// TIA Portal V17 export
// export: Created 2025-03-05T08:01:21.5015692Z, ExportSetting WithDefaults, DisplayName Totally Integrated Automation Portal, DisplayVersion V17 Update 8, DisplayName TIA Portal Openness, DisplayVersion V17 Update 8, DisplayName TIA Portal Version Control Interface, DisplayVersion V17, DisplayName SINAMICS Startdrive Advanced, DisplayVersion V17 SP2, DisplayName SINAMICS Startdrive G110M, G120, G120C, G120D, G120P, G115D, DisplayVersion V17 SP2, DisplayName SINAMICS Startdrive G130, G150, S120, S150, SINAMICS MV, S210, DisplayVersion V17 SP2, DisplayName STEP 7 Professional, DisplayVersion V17 Update 8, DisplayName SINUMERIK ONE STEP 7 Toolbox, DisplayVersion V17 Update 12, DisplayName SINUMERIK 840D sl STEP 7 Toolbox, DisplayVersion V17 Update 12, DisplayName STEP 7 Safety, DisplayVersion V17 Update 6, DisplayName WinCC Advanced, DisplayVersion V17 Update 8
FUNCTION "FC20202_LASER_TRUMPF_ACTIVE" : Void   // FC20202, LAD
TITLE = FC20202 LASER TRUMPF ACTIVE
{ S7_Optimized_Access := 'TRUE' }
VERSION : 0.1
// stored: AutoNumber false, IsIECCheckEnabled false, SetENOAutomatically false, UDAEnableTagReadback false
BEGIN

REGION Network 1: LASER UNIT 1 ACTIVE
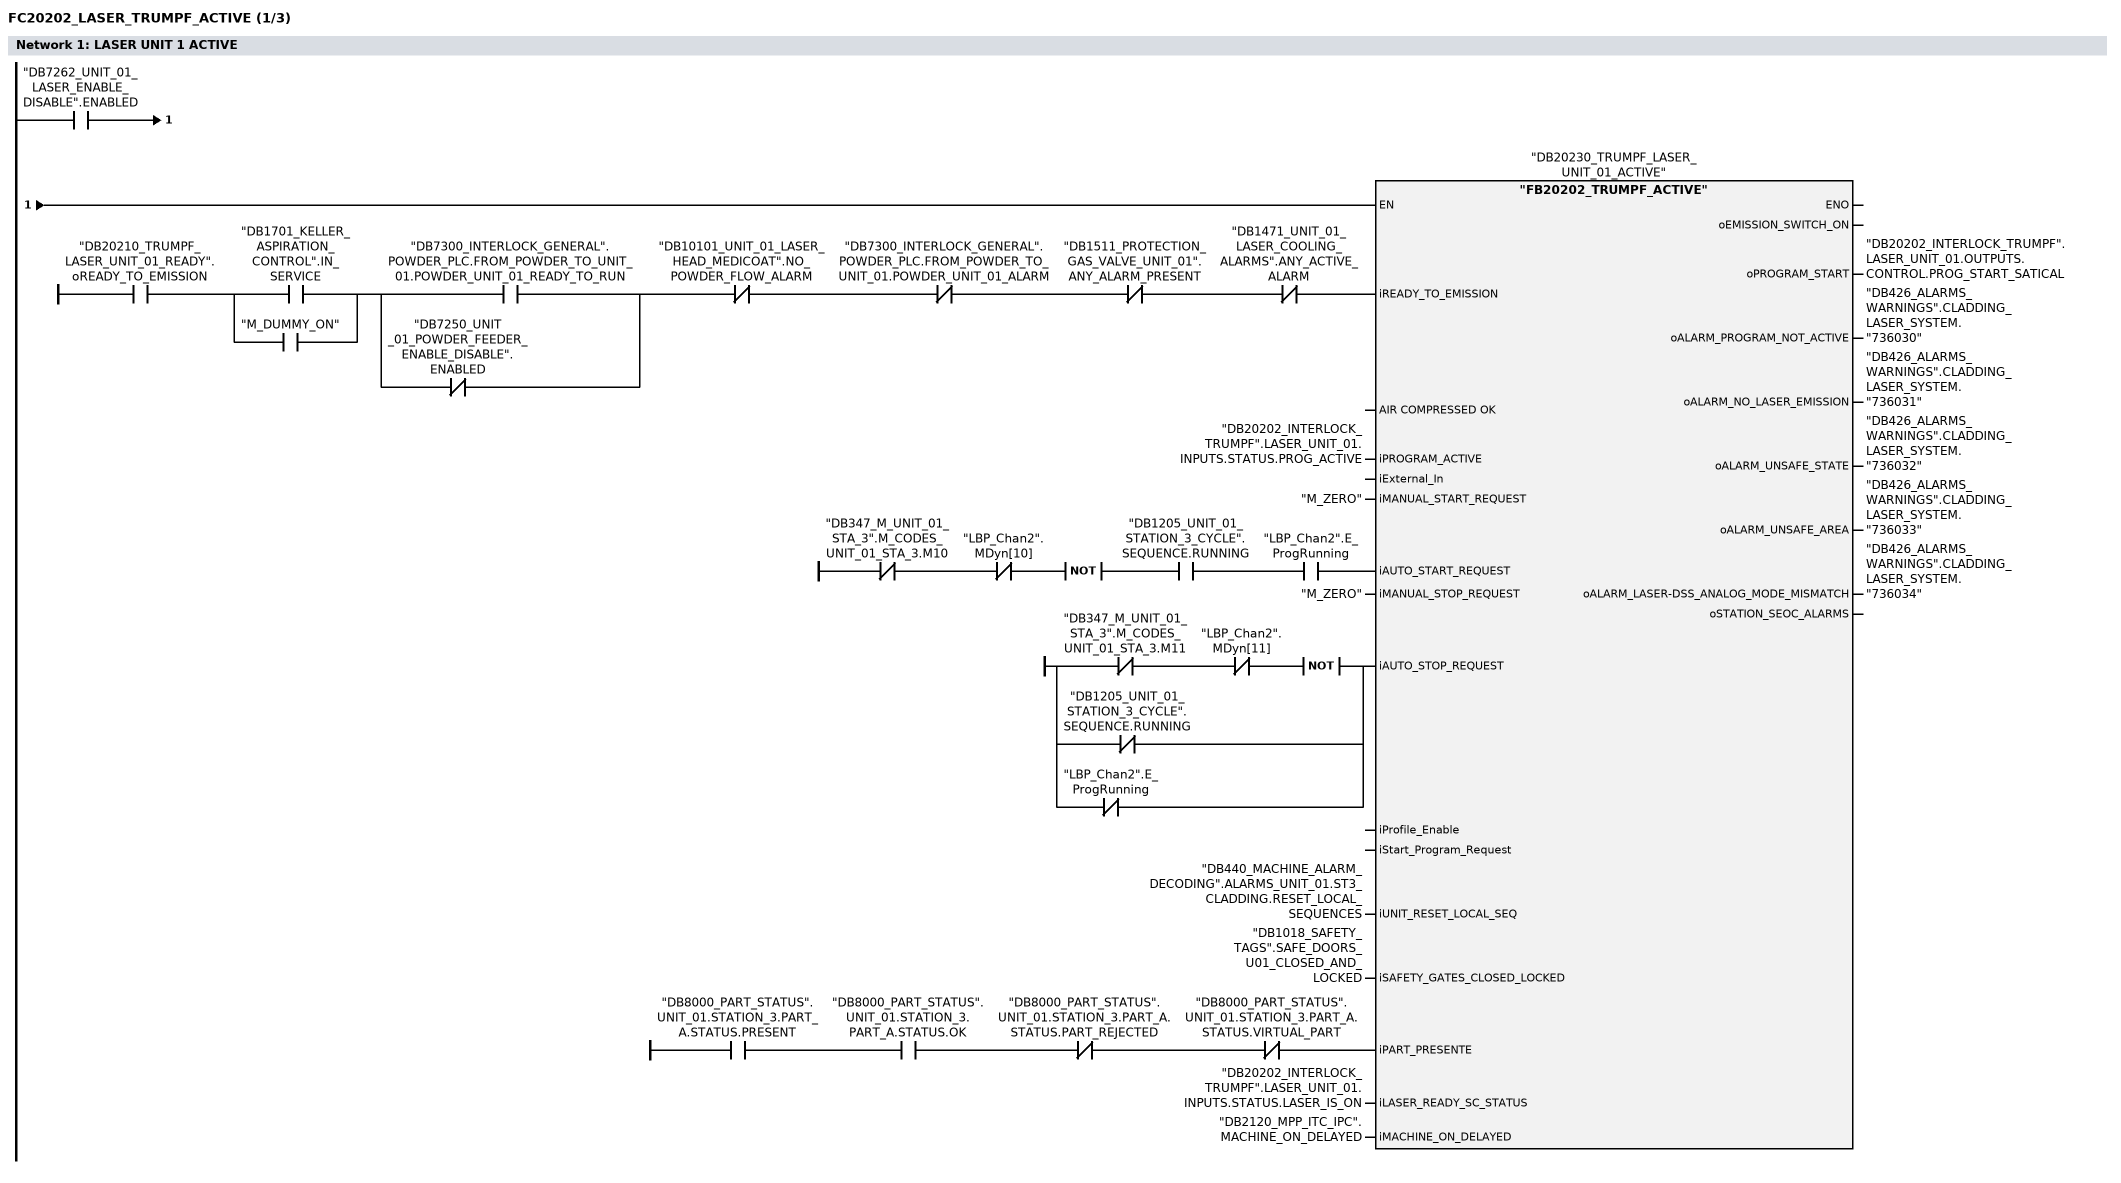
   RUNG wire#powerrail
      Contact( "DB7262_UNIT_01_LASER_ENABLE_DISABLE".ENABLED )
      "DB20230_TRUMPF_LASER_UNIT_01_ACTIVE"(iREADY_TO_EMISSION := wire#w4, iAUTO_START_REQUEST := wire#w5, iAUTO_STOP_REQUEST := wire#w6, iPART_PRESENTE := wire#w7, "AIR COMPRESSED OK" :=, iPROGRAM_ACTIVE := "DB20202_INTERLOCK_TRUMPF".LASER_UNIT_01.INPUTS.STATUS.PROG_ACTIVE, iExternal_In :=, iMANUAL_START_REQUEST := "M_ZERO", iMANUAL_STOP_REQUEST := "M_ZERO", iProfile_Enable :=, iStart_Program_Request :=, iUNIT_RESET_LOCAL_SEQ := "DB440_MACHINE_ALARM_DECODING".ALARMS_UNIT_01.ST3_CLADDING.RESET_LOCAL_SEQUENCES, iSAFETY_GATES_CLOSED_LOCKED := "DB1018_SAFETY_TAGS".SAFE_DOORS_U01_CLOSED_AND_LOCKED, iLASER_READY_SC_STATUS := "DB20202_INTERLOCK_TRUMPF".LASER_UNIT_01.INPUTS.STATUS.LASER_IS_ON, iMACHINE_ON_DELAYED := "DB2120_MPP_ITC_IPC".MACHINE_ON_DELAYED, oEMISSION_SWITCH_ON =>, oPROGRAM_START => "DB20202_INTERLOCK_TRUMPF".LASER_UNIT_01.OUTPUTS.CONTROL.PROG_START_SATICAL, oALARM_PROGRAM_NOT_ACTIVE => "DB426_ALARMS_WARNINGS".CLADDING_LASER_SYSTEM."736030", oALARM_NO_LASER_EMISSION => "DB426_ALARMS_WARNINGS".CLADDING_LASER_SYSTEM."736031", oALARM_UNSAFE_STATE => "DB426_ALARMS_WARNINGS".CLADDING_LASER_SYSTEM."736032", oALARM_UNSAFE_AREA => "DB426_ALARMS_WARNINGS".CLADDING_LASER_SYSTEM."736033", "oALARM_LASER-DSS_ANALOG_MODE_MISMATCH" => "DB426_ALARMS_WARNINGS".CLADDING_LASER_SYSTEM."736034", oSTATION_SEOC_ALARMS =>)
   END_RUNG
   RUNG wire#powerrail
      Contact( "DB20210_TRUMPF_LASER_UNIT_01_READY".oREADY_TO_EMISSION )
      wire#w1
      Contact( "DB1701_KELLER_ASPIRATION_CONTROL".IN_SERVICE )
      wire#w2
      Contact( "DB7300_INTERLOCK_GENERAL".POWDER_PLC.FROM_POWDER_TO_UNIT_01.POWDER_UNIT_01_READY_TO_RUN )
      wire#w3
      I_Contact( "DB10101_UNIT_01_LASER_HEAD_MEDICOAT".NO_POWDER_FLOW_ALARM )
      I_Contact( "DB7300_INTERLOCK_GENERAL".POWDER_PLC.FROM_POWDER_TO_UNIT_01.POWDER_UNIT_01_ALARM )
      I_Contact( "DB1511_PROTECTION_GAS_VALVE_UNIT_01".ANY_ALARM_PRESENT )
      I_Contact( "DB1471_UNIT_01_LASER_COOLING_ALARMS".ANY_ACTIVE_ALARM )
   END_RUNG wire#w4
   RUNG wire#w1
      Contact( "M_DUMMY_ON" )
   END_RUNG wire#w2
   RUNG wire#w2
      I_Contact( "DB7250_UNIT _01_POWDER_FEEDER_ENABLE_DISABLE".ENABLED )
   END_RUNG wire#w3
   RUNG wire#powerrail
      I_Contact( "DB347_M_UNIT_01_STA_3".M_CODES_UNIT_01_STA_3.M10 )
      I_Contact( "LBP_Chan2".MDyn[10] )
      Not()
      Contact( "DB1205_UNIT_01_STATION_3_CYCLE".SEQUENCE.RUNNING )
      Contact( "LBP_Chan2".E_ProgRunning )
   END_RUNG wire#w5
   RUNG wire#powerrail
      I_Contact( "DB347_M_UNIT_01_STA_3".M_CODES_UNIT_01_STA_3.M11 )
      I_Contact( "LBP_Chan2".MDyn[11] )
      Not()
   END_RUNG wire#w6
   RUNG wire#powerrail
      I_Contact( "DB1205_UNIT_01_STATION_3_CYCLE".SEQUENCE.RUNNING )
   END_RUNG wire#w6
   RUNG wire#powerrail
      I_Contact( "LBP_Chan2".E_ProgRunning )
   END_RUNG wire#w6
   RUNG wire#powerrail
      Contact( "DB8000_PART_STATUS".UNIT_01.STATION_3.PART_A.STATUS.PRESENT )
      Contact( "DB8000_PART_STATUS".UNIT_01.STATION_3.PART_A.STATUS.OK )
      I_Contact( "DB8000_PART_STATUS".UNIT_01.STATION_3.PART_A.STATUS.PART_REJECTED )
      I_Contact( "DB8000_PART_STATUS".UNIT_01.STATION_3.PART_A.STATUS.VIRTUAL_PART )
   END_RUNG wire#w7
   // the same network as SCL:
   IF "DB7262_UNIT_01_LASER_ENABLE_DISABLE".ENABLED THEN
       "DB20230_TRUMPF_LASER_UNIT_01_ACTIVE"(iREADY_TO_EMISSION := "DB20210_TRUMPF_LASER_UNIT_01_READY".oREADY_TO_EMISSION AND ("DB1701_KELLER_ASPIRATION_CONTROL".IN_SERVICE OR "M_DUMMY_ON") AND ("DB7300_INTERLOCK_GENERAL".POWDER_PLC.FROM_POWDER_TO_UNIT_01.POWDER_UNIT_01_READY_TO_RUN OR NOT "DB7250_UNIT _01_POWDER_FEEDER_ENABLE_DISABLE".ENABLED) AND NOT "DB10101_UNIT_01_LASER_HEAD_MEDICOAT".NO_POWDER_FLOW_ALARM AND NOT "DB7300_INTERLOCK_GENERAL".POWDER_PLC.FROM_POWDER_TO_UNIT_01.POWDER_UNIT_01_ALARM AND NOT "DB1511_PROTECTION_GAS_VALVE_UNIT_01".ANY_ALARM_PRESENT AND NOT "DB1471_UNIT_01_LASER_COOLING_ALARMS".ANY_ACTIVE_ALARM,   // "FB20202_TRUMPF_ACTIVE"
                               iPROGRAM_ACTIVE := "DB20202_INTERLOCK_TRUMPF".LASER_UNIT_01.INPUTS.STATUS.PROG_ACTIVE,
                               iMANUAL_START_REQUEST := "M_ZERO",
                               iAUTO_START_REQUEST := NOT (NOT "DB347_M_UNIT_01_STA_3".M_CODES_UNIT_01_STA_3.M10 AND NOT "LBP_Chan2".MDyn[10]) AND "DB1205_UNIT_01_STATION_3_CYCLE".SEQUENCE.RUNNING AND "LBP_Chan2".E_ProgRunning,
                               iMANUAL_STOP_REQUEST := "M_ZERO",
                               iAUTO_STOP_REQUEST := NOT (NOT "DB347_M_UNIT_01_STA_3".M_CODES_UNIT_01_STA_3.M11 AND NOT "LBP_Chan2".MDyn[11]) OR NOT "DB1205_UNIT_01_STATION_3_CYCLE".SEQUENCE.RUNNING OR NOT "LBP_Chan2".E_ProgRunning,
                               iUNIT_RESET_LOCAL_SEQ := "DB440_MACHINE_ALARM_DECODING".ALARMS_UNIT_01.ST3_CLADDING.RESET_LOCAL_SEQUENCES,
                               iSAFETY_GATES_CLOSED_LOCKED := "DB1018_SAFETY_TAGS".SAFE_DOORS_U01_CLOSED_AND_LOCKED,
                               iPART_PRESENTE := "DB8000_PART_STATUS".UNIT_01.STATION_3.PART_A.STATUS.PRESENT AND "DB8000_PART_STATUS".UNIT_01.STATION_3.PART_A.STATUS.OK AND NOT "DB8000_PART_STATUS".UNIT_01.STATION_3.PART_A.STATUS.PART_REJECTED AND NOT "DB8000_PART_STATUS".UNIT_01.STATION_3.PART_A.STATUS.VIRTUAL_PART,
                               iLASER_READY_SC_STATUS := "DB20202_INTERLOCK_TRUMPF".LASER_UNIT_01.INPUTS.STATUS.LASER_IS_ON,
                               iMACHINE_ON_DELAYED := "DB2120_MPP_ITC_IPC".MACHINE_ON_DELAYED,
                               oPROGRAM_START => "DB20202_INTERLOCK_TRUMPF".LASER_UNIT_01.OUTPUTS.CONTROL.PROG_START_SATICAL,
                               oALARM_PROGRAM_NOT_ACTIVE => "DB426_ALARMS_WARNINGS".CLADDING_LASER_SYSTEM."736030",
                               oALARM_NO_LASER_EMISSION => "DB426_ALARMS_WARNINGS".CLADDING_LASER_SYSTEM."736031",
                               oALARM_UNSAFE_STATE => "DB426_ALARMS_WARNINGS".CLADDING_LASER_SYSTEM."736032",
                               oALARM_UNSAFE_AREA => "DB426_ALARMS_WARNINGS".CLADDING_LASER_SYSTEM."736033",
                               "oALARM_LASER-DSS_ANALOG_MODE_MISMATCH" => "DB426_ALARMS_WARNINGS".CLADDING_LASER_SYSTEM."736034");
   END_IF;
END_REGION

REGION Network 2: LASER UNIT 2 ACTIVE
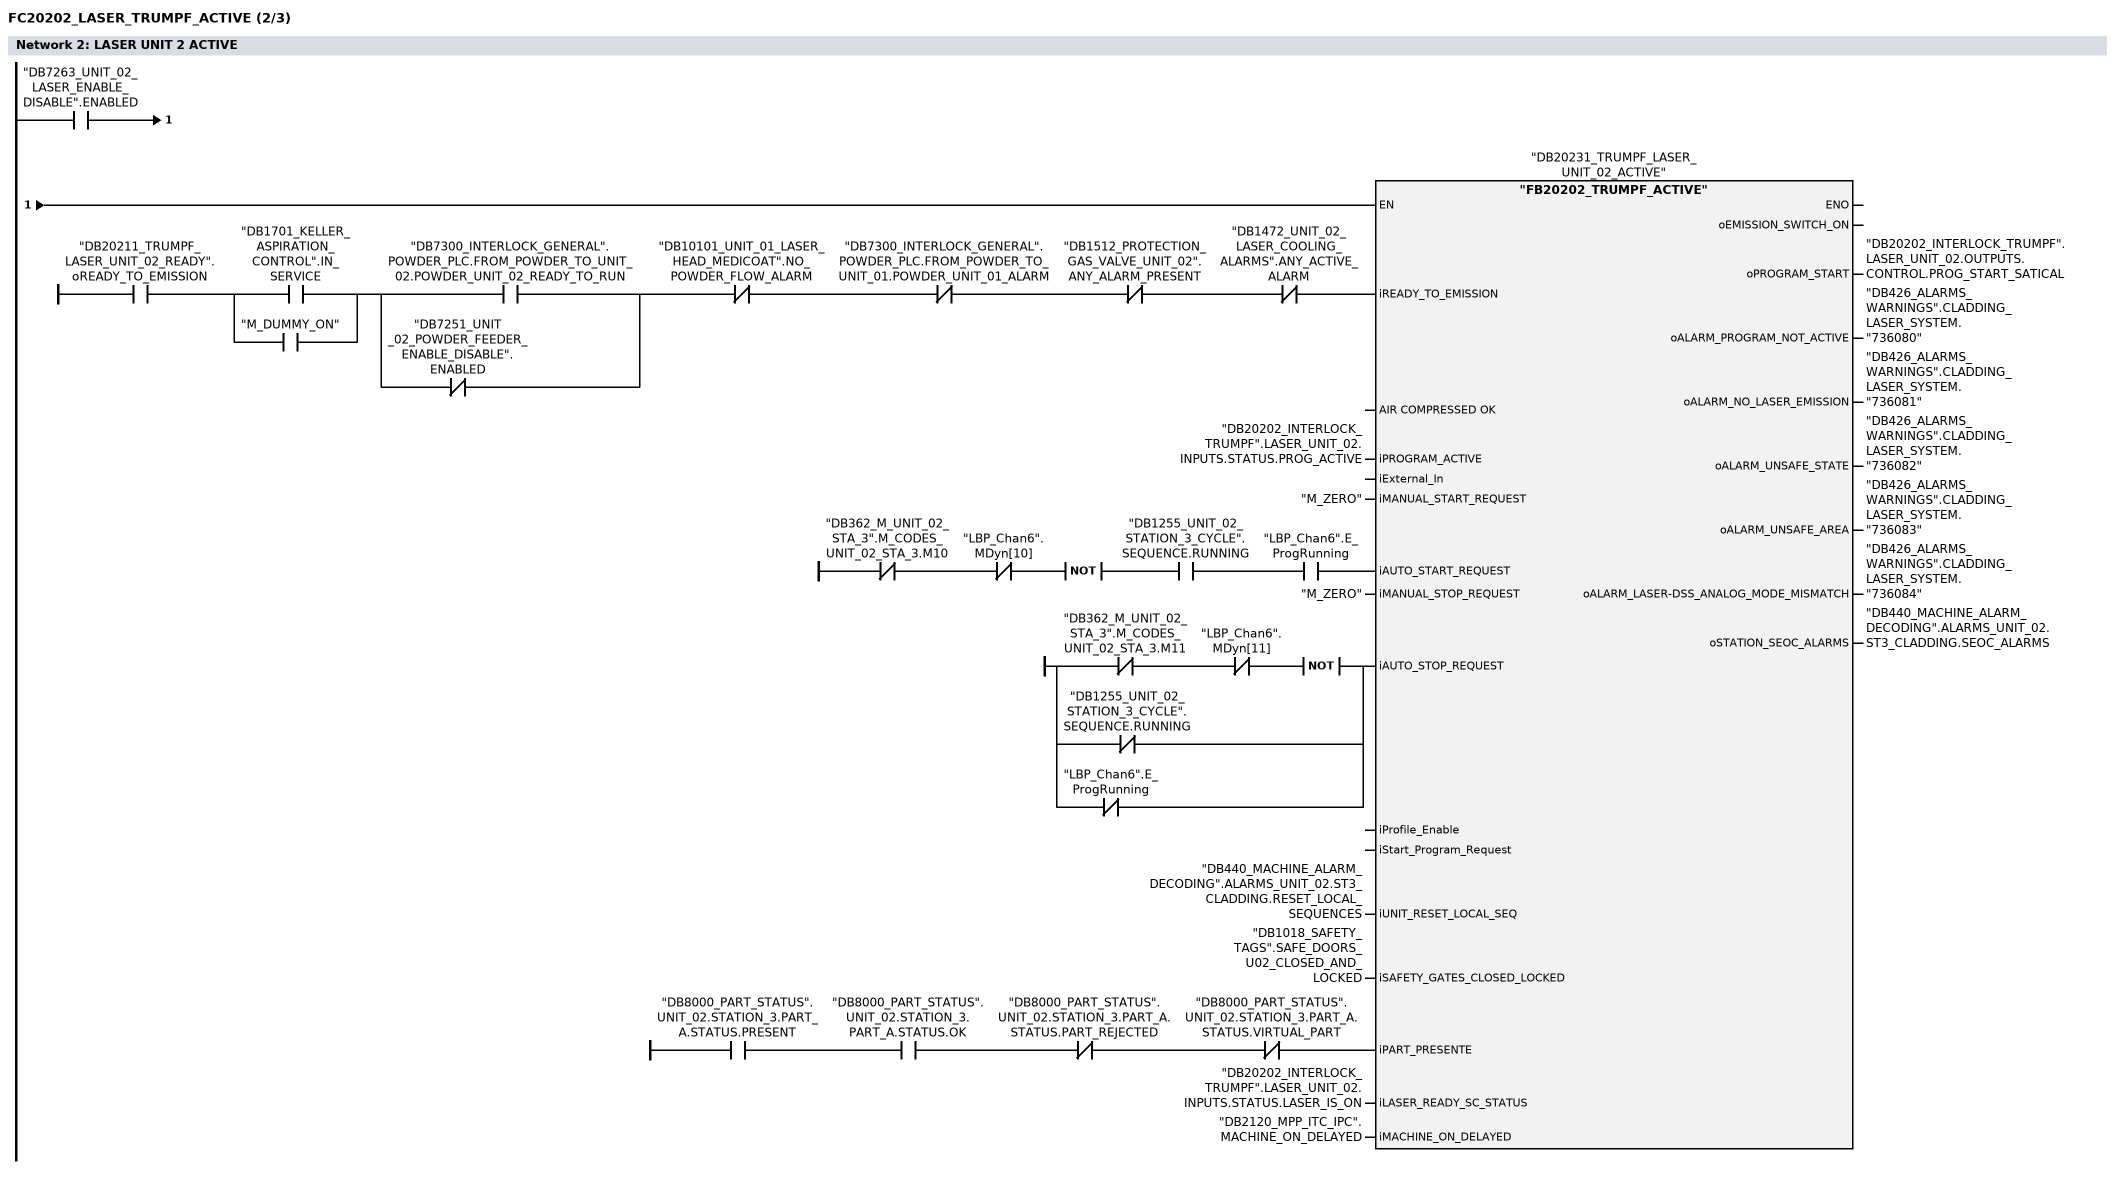
   RUNG wire#powerrail
      Contact( "DB7263_UNIT_02_LASER_ENABLE_DISABLE".ENABLED )
      "DB20231_TRUMPF_LASER_UNIT_02_ACTIVE"(iREADY_TO_EMISSION := wire#w4, iAUTO_START_REQUEST := wire#w5, iAUTO_STOP_REQUEST := wire#w6, iPART_PRESENTE := wire#w7, "AIR COMPRESSED OK" :=, iPROGRAM_ACTIVE := "DB20202_INTERLOCK_TRUMPF".LASER_UNIT_02.INPUTS.STATUS.PROG_ACTIVE, iExternal_In :=, iMANUAL_START_REQUEST := "M_ZERO", iMANUAL_STOP_REQUEST := "M_ZERO", iProfile_Enable :=, iStart_Program_Request :=, iUNIT_RESET_LOCAL_SEQ := "DB440_MACHINE_ALARM_DECODING".ALARMS_UNIT_02.ST3_CLADDING.RESET_LOCAL_SEQUENCES, iSAFETY_GATES_CLOSED_LOCKED := "DB1018_SAFETY_TAGS".SAFE_DOORS_U02_CLOSED_AND_LOCKED, iLASER_READY_SC_STATUS := "DB20202_INTERLOCK_TRUMPF".LASER_UNIT_02.INPUTS.STATUS.LASER_IS_ON, iMACHINE_ON_DELAYED := "DB2120_MPP_ITC_IPC".MACHINE_ON_DELAYED, oEMISSION_SWITCH_ON =>, oPROGRAM_START => "DB20202_INTERLOCK_TRUMPF".LASER_UNIT_02.OUTPUTS.CONTROL.PROG_START_SATICAL, oALARM_PROGRAM_NOT_ACTIVE => "DB426_ALARMS_WARNINGS".CLADDING_LASER_SYSTEM."736080", oALARM_NO_LASER_EMISSION => "DB426_ALARMS_WARNINGS".CLADDING_LASER_SYSTEM."736081", oALARM_UNSAFE_STATE => "DB426_ALARMS_WARNINGS".CLADDING_LASER_SYSTEM."736082", oALARM_UNSAFE_AREA => "DB426_ALARMS_WARNINGS".CLADDING_LASER_SYSTEM."736083", "oALARM_LASER-DSS_ANALOG_MODE_MISMATCH" => "DB426_ALARMS_WARNINGS".CLADDING_LASER_SYSTEM."736084", oSTATION_SEOC_ALARMS => "DB440_MACHINE_ALARM_DECODING".ALARMS_UNIT_02.ST3_CLADDING.SEOC_ALARMS)
   END_RUNG
   RUNG wire#powerrail
      Contact( "DB20211_TRUMPF_LASER_UNIT_02_READY".oREADY_TO_EMISSION )
      wire#w1
      Contact( "DB1701_KELLER_ASPIRATION_CONTROL".IN_SERVICE )
      wire#w2
      Contact( "DB7300_INTERLOCK_GENERAL".POWDER_PLC.FROM_POWDER_TO_UNIT_02.POWDER_UNIT_02_READY_TO_RUN )
      wire#w3
      I_Contact( "DB10101_UNIT_01_LASER_HEAD_MEDICOAT".NO_POWDER_FLOW_ALARM )
      I_Contact( "DB7300_INTERLOCK_GENERAL".POWDER_PLC.FROM_POWDER_TO_UNIT_01.POWDER_UNIT_01_ALARM )
      I_Contact( "DB1512_PROTECTION_GAS_VALVE_UNIT_02".ANY_ALARM_PRESENT )
      I_Contact( "DB1472_UNIT_02_LASER_COOLING_ALARMS".ANY_ACTIVE_ALARM )
   END_RUNG wire#w4
   RUNG wire#w1
      Contact( "M_DUMMY_ON" )
   END_RUNG wire#w2
   RUNG wire#w2
      I_Contact( "DB7251_UNIT _02_POWDER_FEEDER_ENABLE_DISABLE".ENABLED )
   END_RUNG wire#w3
   RUNG wire#powerrail
      I_Contact( "DB362_M_UNIT_02_STA_3".M_CODES_UNIT_02_STA_3.M10 )
      I_Contact( "LBP_Chan6".MDyn[10] )
      Not()
      Contact( "DB1255_UNIT_02_STATION_3_CYCLE".SEQUENCE.RUNNING )
      Contact( "LBP_Chan6".E_ProgRunning )
   END_RUNG wire#w5
   RUNG wire#powerrail
      I_Contact( "DB362_M_UNIT_02_STA_3".M_CODES_UNIT_02_STA_3.M11 )
      I_Contact( "LBP_Chan6".MDyn[11] )
      Not()
   END_RUNG wire#w6
   RUNG wire#powerrail
      I_Contact( "DB1255_UNIT_02_STATION_3_CYCLE".SEQUENCE.RUNNING )
   END_RUNG wire#w6
   RUNG wire#powerrail
      I_Contact( "LBP_Chan6".E_ProgRunning )
   END_RUNG wire#w6
   RUNG wire#powerrail
      Contact( "DB8000_PART_STATUS".UNIT_02.STATION_3.PART_A.STATUS.PRESENT )
      Contact( "DB8000_PART_STATUS".UNIT_02.STATION_3.PART_A.STATUS.OK )
      I_Contact( "DB8000_PART_STATUS".UNIT_02.STATION_3.PART_A.STATUS.PART_REJECTED )
      I_Contact( "DB8000_PART_STATUS".UNIT_02.STATION_3.PART_A.STATUS.VIRTUAL_PART )
   END_RUNG wire#w7
   // the same network as SCL:
   IF "DB7263_UNIT_02_LASER_ENABLE_DISABLE".ENABLED THEN
       "DB20231_TRUMPF_LASER_UNIT_02_ACTIVE"(iREADY_TO_EMISSION := "DB20211_TRUMPF_LASER_UNIT_02_READY".oREADY_TO_EMISSION AND ("DB1701_KELLER_ASPIRATION_CONTROL".IN_SERVICE OR "M_DUMMY_ON") AND ("DB7300_INTERLOCK_GENERAL".POWDER_PLC.FROM_POWDER_TO_UNIT_02.POWDER_UNIT_02_READY_TO_RUN OR NOT "DB7251_UNIT _02_POWDER_FEEDER_ENABLE_DISABLE".ENABLED) AND NOT "DB10101_UNIT_01_LASER_HEAD_MEDICOAT".NO_POWDER_FLOW_ALARM AND NOT "DB7300_INTERLOCK_GENERAL".POWDER_PLC.FROM_POWDER_TO_UNIT_01.POWDER_UNIT_01_ALARM AND NOT "DB1512_PROTECTION_GAS_VALVE_UNIT_02".ANY_ALARM_PRESENT AND NOT "DB1472_UNIT_02_LASER_COOLING_ALARMS".ANY_ACTIVE_ALARM,   // "FB20202_TRUMPF_ACTIVE"
                               iPROGRAM_ACTIVE := "DB20202_INTERLOCK_TRUMPF".LASER_UNIT_02.INPUTS.STATUS.PROG_ACTIVE,
                               iMANUAL_START_REQUEST := "M_ZERO",
                               iAUTO_START_REQUEST := NOT (NOT "DB362_M_UNIT_02_STA_3".M_CODES_UNIT_02_STA_3.M10 AND NOT "LBP_Chan6".MDyn[10]) AND "DB1255_UNIT_02_STATION_3_CYCLE".SEQUENCE.RUNNING AND "LBP_Chan6".E_ProgRunning,
                               iMANUAL_STOP_REQUEST := "M_ZERO",
                               iAUTO_STOP_REQUEST := NOT (NOT "DB362_M_UNIT_02_STA_3".M_CODES_UNIT_02_STA_3.M11 AND NOT "LBP_Chan6".MDyn[11]) OR NOT "DB1255_UNIT_02_STATION_3_CYCLE".SEQUENCE.RUNNING OR NOT "LBP_Chan6".E_ProgRunning,
                               iUNIT_RESET_LOCAL_SEQ := "DB440_MACHINE_ALARM_DECODING".ALARMS_UNIT_02.ST3_CLADDING.RESET_LOCAL_SEQUENCES,
                               iSAFETY_GATES_CLOSED_LOCKED := "DB1018_SAFETY_TAGS".SAFE_DOORS_U02_CLOSED_AND_LOCKED,
                               iPART_PRESENTE := "DB8000_PART_STATUS".UNIT_02.STATION_3.PART_A.STATUS.PRESENT AND "DB8000_PART_STATUS".UNIT_02.STATION_3.PART_A.STATUS.OK AND NOT "DB8000_PART_STATUS".UNIT_02.STATION_3.PART_A.STATUS.PART_REJECTED AND NOT "DB8000_PART_STATUS".UNIT_02.STATION_3.PART_A.STATUS.VIRTUAL_PART,
                               iLASER_READY_SC_STATUS := "DB20202_INTERLOCK_TRUMPF".LASER_UNIT_02.INPUTS.STATUS.LASER_IS_ON,
                               iMACHINE_ON_DELAYED := "DB2120_MPP_ITC_IPC".MACHINE_ON_DELAYED,
                               oPROGRAM_START => "DB20202_INTERLOCK_TRUMPF".LASER_UNIT_02.OUTPUTS.CONTROL.PROG_START_SATICAL,
                               oALARM_PROGRAM_NOT_ACTIVE => "DB426_ALARMS_WARNINGS".CLADDING_LASER_SYSTEM."736080",
                               oALARM_NO_LASER_EMISSION => "DB426_ALARMS_WARNINGS".CLADDING_LASER_SYSTEM."736081",
                               oALARM_UNSAFE_STATE => "DB426_ALARMS_WARNINGS".CLADDING_LASER_SYSTEM."736082",
                               oALARM_UNSAFE_AREA => "DB426_ALARMS_WARNINGS".CLADDING_LASER_SYSTEM."736083",
                               "oALARM_LASER-DSS_ANALOG_MODE_MISMATCH" => "DB426_ALARMS_WARNINGS".CLADDING_LASER_SYSTEM."736084",
                               oSTATION_SEOC_ALARMS => "DB440_MACHINE_ALARM_DECODING".ALARMS_UNIT_02.ST3_CLADDING.SEOC_ALARMS);
   END_IF;
END_REGION

REGION Network 3: AXIS FROM UNIT 01 NOT MOVING WHILE LASER ON FAULT
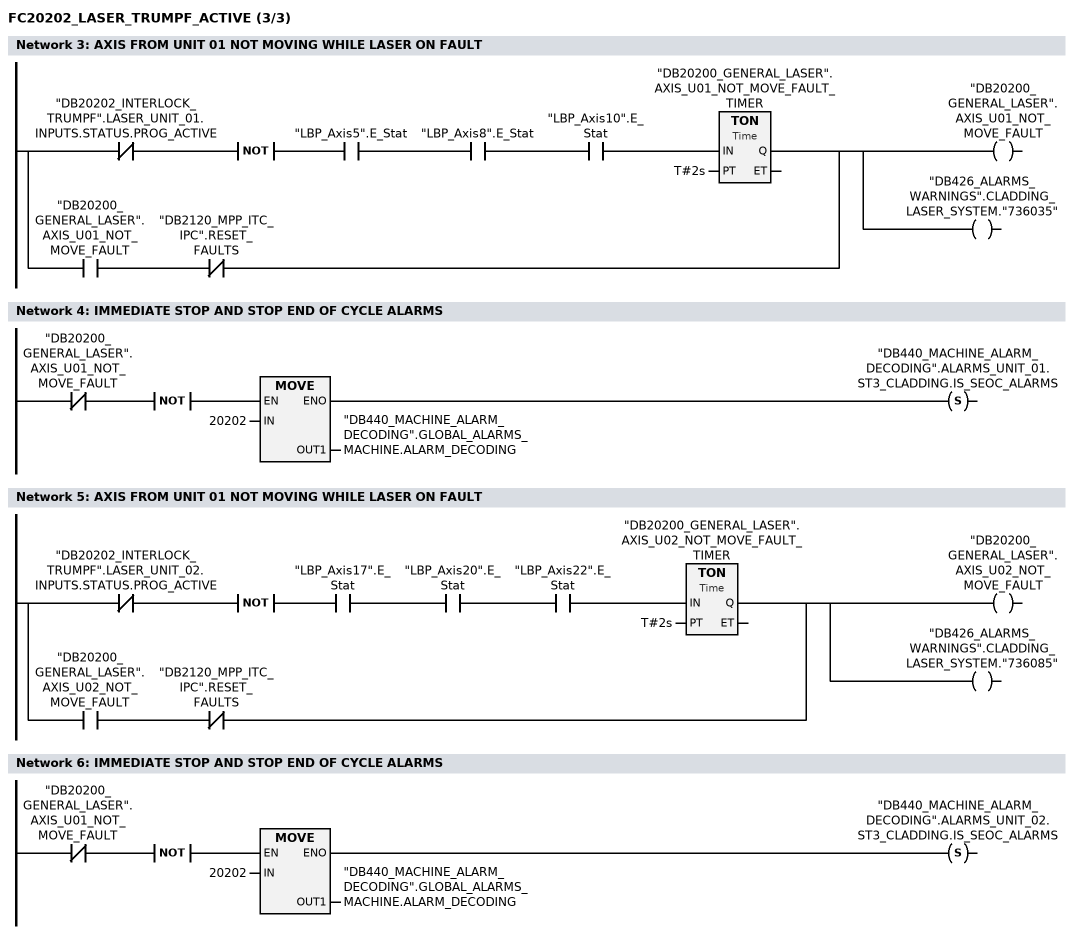
   RUNG wire#powerrail
      I_Contact( "DB20202_INTERLOCK_TRUMPF".LASER_UNIT_01.INPUTS.STATUS.PROG_ACTIVE )
      Not()
      Contact( "LBP_Axis5".E_Stat )
      Contact( "LBP_Axis8".E_Stat )
      Contact( "LBP_Axis10".E_Stat )
      { S7_Templates := "time_type := Time" } "DB20200_GENERAL_LASER".AXIS_U01_NOT_MOVE_FAULT_TIMER.TON(pt := T#2s, et =>)
      wire#w1
      Coil( "DB20200_GENERAL_LASER".AXIS_U01_NOT_MOVE_FAULT )
   END_RUNG
   RUNG wire#powerrail
      Contact( "DB20200_GENERAL_LASER".AXIS_U01_NOT_MOVE_FAULT )
      I_Contact( "DB2120_MPP_ITC_IPC".RESET_FAULTS )
   END_RUNG wire#w1
   RUNG wire#w1
      Coil( "DB426_ALARMS_WARNINGS".CLADDING_LASER_SYSTEM."736035" )
   END_RUNG
   // the same network as SCL:
   "DB20200_GENERAL_LASER".AXIS_U01_NOT_MOVE_FAULT_TIMER.TON(IN := NOT (NOT "DB20202_INTERLOCK_TRUMPF".LASER_UNIT_01.INPUTS.STATUS.PROG_ACTIVE) AND "LBP_Axis5".E_Stat AND "LBP_Axis8".E_Stat AND "LBP_Axis10".E_Stat,
                           PT := T#2s);
   "DB20200_GENERAL_LASER".AXIS_U01_NOT_MOVE_FAULT := "DB20200_GENERAL_LASER".AXIS_U01_NOT_MOVE_FAULT_TIMER.Q OR ("DB20200_GENERAL_LASER".AXIS_U01_NOT_MOVE_FAULT AND NOT "DB2120_MPP_ITC_IPC".RESET_FAULTS);
   "DB426_ALARMS_WARNINGS".CLADDING_LASER_SYSTEM."736035" := "DB20200_GENERAL_LASER".AXIS_U01_NOT_MOVE_FAULT;
END_REGION

REGION Network 4: IMMEDIATE STOP AND STOP END OF CYCLE ALARMS
   RUNG wire#powerrail
      I_Contact( "DB20200_GENERAL_LASER".AXIS_U01_NOT_MOVE_FAULT )
      Not()
      Move(in := 20202, out1 => "DB440_MACHINE_ALARM_DECODING".GLOBAL_ALARMS_MACHINE.ALARM_DECODING)
      S_Coil( "DB440_MACHINE_ALARM_DECODING".ALARMS_UNIT_01.ST3_CLADDING.IS_SEOC_ALARMS )
   END_RUNG
   // the same network as SCL:
   IF NOT (NOT "DB20200_GENERAL_LASER".AXIS_U01_NOT_MOVE_FAULT) THEN
       "DB440_MACHINE_ALARM_DECODING".GLOBAL_ALARMS_MACHINE.ALARM_DECODING := 20202;
       "DB440_MACHINE_ALARM_DECODING".ALARMS_UNIT_01.ST3_CLADDING.IS_SEOC_ALARMS := TRUE;
   END_IF;
END_REGION

REGION Network 5: AXIS FROM UNIT 01 NOT MOVING WHILE LASER ON FAULT
   RUNG wire#powerrail
      I_Contact( "DB20202_INTERLOCK_TRUMPF".LASER_UNIT_02.INPUTS.STATUS.PROG_ACTIVE )
      Not()
      Contact( "LBP_Axis17".E_Stat )
      Contact( "LBP_Axis20".E_Stat )
      Contact( "LBP_Axis22".E_Stat )
      { S7_Templates := "time_type := Time" } "DB20200_GENERAL_LASER".AXIS_U02_NOT_MOVE_FAULT_TIMER.TON(pt := T#2s, et =>)
      wire#w1
      Coil( "DB20200_GENERAL_LASER".AXIS_U02_NOT_MOVE_FAULT )
   END_RUNG
   RUNG wire#powerrail
      Contact( "DB20200_GENERAL_LASER".AXIS_U02_NOT_MOVE_FAULT )
      I_Contact( "DB2120_MPP_ITC_IPC".RESET_FAULTS )
   END_RUNG wire#w1
   RUNG wire#w1
      Coil( "DB426_ALARMS_WARNINGS".CLADDING_LASER_SYSTEM."736085" )
   END_RUNG
   // the same network as SCL:
   "DB20200_GENERAL_LASER".AXIS_U02_NOT_MOVE_FAULT_TIMER.TON(IN := NOT (NOT "DB20202_INTERLOCK_TRUMPF".LASER_UNIT_02.INPUTS.STATUS.PROG_ACTIVE) AND "LBP_Axis17".E_Stat AND "LBP_Axis20".E_Stat AND "LBP_Axis22".E_Stat,
                           PT := T#2s);
   "DB20200_GENERAL_LASER".AXIS_U02_NOT_MOVE_FAULT := "DB20200_GENERAL_LASER".AXIS_U02_NOT_MOVE_FAULT_TIMER.Q OR ("DB20200_GENERAL_LASER".AXIS_U02_NOT_MOVE_FAULT AND NOT "DB2120_MPP_ITC_IPC".RESET_FAULTS);
   "DB426_ALARMS_WARNINGS".CLADDING_LASER_SYSTEM."736085" := "DB20200_GENERAL_LASER".AXIS_U02_NOT_MOVE_FAULT;
END_REGION

REGION Network 6: IMMEDIATE STOP AND STOP END OF CYCLE ALARMS
   RUNG wire#powerrail
      I_Contact( "DB20200_GENERAL_LASER".AXIS_U01_NOT_MOVE_FAULT )
      Not()
      Move(in := 20202, out1 => "DB440_MACHINE_ALARM_DECODING".GLOBAL_ALARMS_MACHINE.ALARM_DECODING)
      S_Coil( "DB440_MACHINE_ALARM_DECODING".ALARMS_UNIT_02.ST3_CLADDING.IS_SEOC_ALARMS )
   END_RUNG
   // the same network as SCL:
   IF NOT (NOT "DB20200_GENERAL_LASER".AXIS_U01_NOT_MOVE_FAULT) THEN
       "DB440_MACHINE_ALARM_DECODING".GLOBAL_ALARMS_MACHINE.ALARM_DECODING := 20202;
       "DB440_MACHINE_ALARM_DECODING".ALARMS_UNIT_02.ST3_CLADDING.IS_SEOC_ALARMS := TRUE;
   END_IF;
END_REGION
END_FUNCTION
